Fanuc KAREL source: kt00222.KL

-- PROVISIONAL review KL for V770-1; original PC SHA256 971d86cc0f43f5b8753882d3b470d83a786b82bbecd91dbd77c36c296385ba3a
-- Incomplete behavior may be omitted. Consult companion uncertainty JSON. Do not deploy.
PROGRAM KT00222
%NOLOCKGROUP
VAR
  OUT : INTEGER
-- UNRESOLVED_DECL H1 type=002017
-- UNRESOLVED_DECL Y2 type=002018
BEGIN
  -- UNRESOLVED_PC offsets 5-19; opcodes 2E,22,9D,33,B4
  -- UNRESOLVED_PC offsets 24-38; opcodes 2E,22,9D,33,B2
  -- UNRESOLVED_PC offsets 43-68; opcodes 22,9D,33,B3,22,9D,33,B1,46,23
  -- UNRESOLVED_PC offsets 73-77; opcodes 7F
END KT00222
